DATA_BLOCK "DB_PlcSessionStatus"
{ S7_Optimized_Access := 'TRUE' }
VERSION : 0.1
NON_RETAIN
   VAR
      Data : "UDT_PlcSessionStatus";
   END_VAR

BEGIN
END_DATA_BLOCK
